// TIA Portal V18 export
FUNCTION_BLOCK "flow_measurement"   // FB5, LAD
{ S7_Optimized_Access := 'TRUE' }
VERSION : 0.1
// stored: AutoNumber true, IsIECCheckEnabled false, IsRetainMemResEnabled false, MemoryReserve 100, SetENOAutomatically false, UDAEnableTagReadback false
   VAR
      K_factor : Real := 10.0;
   END_VAR
   VAR_TEMP
      Done : Bool;
      Busy : Bool;
      error : Bool;
      status : Word;
      pulse1_Temp : DInt;
      cv1 : Int;
   END_VAR
BEGIN

REGION Network 1: To simulate the Pulses from flow meter
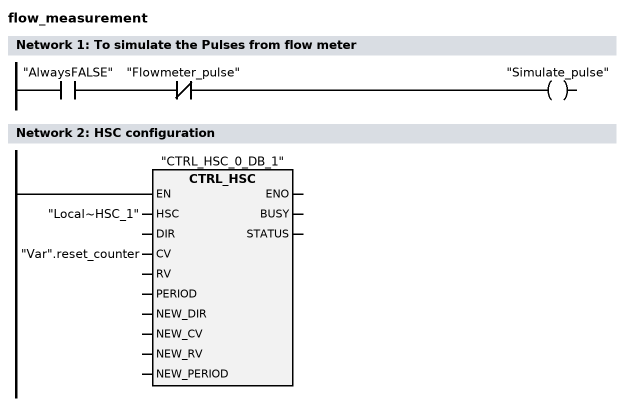
   RUNG wire#powerrail
      Contact( "AlwaysFALSE" )
      I_Contact( "Flowmeter_pulse" )
      Coil( "Simulate_pulse" )
   END_RUNG
   // the same network as SCL:
   "Simulate_pulse" := "AlwaysFALSE" AND NOT "Flowmeter_pulse";
END_REGION

REGION Network 2: HSC configuration
   RUNG wire#powerrail
      "CTRL_HSC_0_DB_1".CTRL_HSC(HSC := "Local~HSC_1", DIR :=, CV := "Var".reset_counter, RV :=, PERIOD :=, NEW_DIR :=, NEW_CV :=, NEW_RV :=, NEW_PERIOD :=, BUSY =>, STATUS =>)
   END_RUNG
   // the same network as SCL:
   "CTRL_HSC_0_DB_1"(HSC := "Local~HSC_1", CV := "Var".reset_counter);   // CTRL_HSC
END_REGION

REGION Network 3 (SCL): Read the value of the counter and put it in the Quantity value


   //counted pulse by HSC
   "Var".counter := "Pulse1";
   "Var".counter_real := DINT_TO_REAL(IN := "Var".counter);



   //K_factor should be edited correctly
   "Var".loaded_quantity := #K_factor * "Pulse1";



   //Time remained(in seconds, that's why multiplied by 3600)
   "Var".remained_quantity := ("Var".set_quantity - REAL_TO_INT("Var".loaded_quantity));
   "Var".time_remained := ("Var".remained_quantity / "Var".instat_flowrate) * 3600;
END_REGION

REGION Network 4 (SCL): Computing the recent loaded quantity (whenever pump starts)


   IF "Var".no_flow_states THEN
       "Var".pulse_temp := "Pulse1";
   END_IF;

   "Var".recent_loaded_quantity := ("Pulse1" - "Var".pulse_temp)* #K_factor;
END_REGION
END_FUNCTION_BLOCK
